// TIA Portal V18 export
// export: Created 2026-06-08T13:24:12.8198007Z, ExportSetting WithDefaults, DisplayName Totally Integrated Automation Portal, DisplayVersion V18, DisplayName TIA Portal Openness, DisplayVersion V18, DisplayName TIA Portal Version Control Interface, DisplayVersion V18, DisplayName STEP 7 Professional, DisplayVersion V18, DisplayName STEP 7 Safety, DisplayVersion V18, DisplayName WinCC Professional, DisplayVersion V18
DATA_BLOCK "DB_Modbus_Holding_Register_DB"   // DB20
TITLE = DB_Modbus_Holding_Register_DB
{ S7_Optimized_Access := 'FALSE' }
VERSION : 0.1
// DB communication via Modbus TCP
// stored: AutoNumber false, DBAccessibleFromOPCUA true, IsOnlyStoredInLoadMemory false, IsWriteProtectedInAS false
   VAR
      CmdSeq : Int;
      Cmd_Start : Bool;
      Cmd_Stop : Bool;
      Cmd_Reset : Bool;
      Cmd_EStop : Bool;
      Cmd_Pump_Branch2_To_SubTanks : Bool;
      Cmd_Load_Recipe : Bool;
      Heartbeat_Client : Int;
      AckSeq : Int;
      Done_Branch2 : Bool;
      Done_Recipe : Bool;
      Alarm : Bool;
      State : Int;
      PID_Bon4_SP : Real;
      PID_Bon4_PV : Real;
      PID_Bon4_CV : Real;
      Heartbeat_Server : Int;
   END_VAR
BEGIN
END_DATA_BLOCK
